# EPICS substitutions: src/iocdoc/testfiles/iocBoot/ioc495idc/templates/xradiaAliases.substitutions
file "$(TOP)/495idcApp/Db/xradia_motorAliases.db"
{
pattern
{P           M,    PA	       MA}

{495idcxxx:,  m1,   495idcnpi:,  m1}
{495idcxxx:,  m2,   495idcnpi:,  m2}
{495idcxxx:,  m3,   495idcnpi:,  m3}
{495idcxxx:,  m4,   495idcnpi:,  m4}
{495idcxxx:,  m5,   495idcnpi:,  m5}
{495idcxxx:,  m6,   495idcnpi:,  m6}
{495idcxxx:,  m7,   495idcnpi:,  m7}
{495idcxxx:,  m8,   495idcnpi:,  m8}
{495idcxxx:,  m9,   495idcnpi:,  m9}
{495idcxxx:,  m10,  495idcnpi:,  m10}
{495idcxxx:,  m11,  495idcnpi:,  m11}
{495idcxxx:,  m12,  495idcnpi:,  m12}
{495idcxxx:,  m13,  495idcnpi:,  m13}
{495idcxxx:,  m14,  495idcnpi:,  m14}
{495idcxxx:,  m15,  495idcnpi:,  m15}
{495idcxxx:,  m16,  495idcnpi:,  m16}
{495idcxxx:,  m17,  495idcnpi:,  m17}
{495idcxxx:,  m18,  495idcnpi:,  m18}
{495idcxxx:,  m19,  495idcnpi:,  m19}
{495idcxxx:,  m20,  495idcnpi:,  m20}
{495idcxxx:,  m21,  495idcnpi:,  m21}
{495idcxxx:,  m22,  495idcnpi:,  m22}
{495idcxxx:,  m23,  495idcnpi:,  m23}
{495idcxxx:,  m24,  495idcnpi:,  m24}
{495idcxxx:,  m25,  495idcnpi:,  m25}
{495idcxxx:,  m26,  495idcnpi:,  m26}
{495idcxxx:,  m27,  495idcnpi:,  m27}
{495idcxxx:,  m28,  495idcnpi:,  m28}
{495idcxxx:,  m29,  495idcnpi:,  m29}

{495idcxxx:,  m34,  495idcnpi:,  m34}
{495idcxxx:,  m35,  495idcnpi:,  m35}

}
